FUNCTION_BLOCK FB_WriteRFID
VAR_INPUT
	bAutoNumber				:BOOL;		
	byFirstByteInput		:BYTE;
	bySecondByteInput		:BYTE;
	byLastByteInput			:BYTE;

	bReset					:BOOL;		//reset licznika
END_VAR
VAR_IN_OUT
	bEnable					:BOOL;		//zalczenie bloku
	byIDtoWrite				:BYTE;		//ID do wczytania
END_VAR


VAR_OUTPUT
	byFirstByteOutput		:BYTE;
	bySecondByteOutput		:BYTE;
	byThirdByteOutput		:BYTE;
	byFourthByteOutput		:BYTE;
	byFifthByteOutput		:BYTE;
	byLastByteOutput		:BYTE;
	bDone					:BOOL;		//informacja o prawidlowym zakoczeniu zapisu
	bError					:BOOL;
	iCounterDone			:INT;		//licznik operacji zapisu zakonczonych sukcesem
END_VAR
VAR
	
	iStep: INT;
	tonDelayError	:TON;
END_VAR

IF bReset THEN
	iCounterDone	:=0;
	iStep := 0;
	byFirstByteOutput := byLastByteOutput := 0;
	bReset := FALSE;
END_IF

CASE iStep OF
	0:  //init	
		IF byFirstByteInput = 129 AND bEnable THEN
			bDone:=FALSE; 
			iStep:=10;
		END_IF
	
	10:  //write command
		bySecondByteOutput 	:= 02;
		byThirdByteOutput	:= 00;
		byFourthByteOutput	:= 00;
		byFifthByteOutput 	:= 01;
		byFirstByteOutput := byLastByteOutput := 01;
	
		IF byFirstByteInput = 163 THEN
			iStep := 20;
		ELSIF NOT byFirstByteInput = 163 AND tonDelayError.Q = TRUE THEN
			iStep := 100;
		END_IF
	
	20: //write data
		IF bAutoNumber THEN
			bySecondByteOutput := byIDtoWrite + INT_TO_BYTE(iCounterDone); 
		ELSE
			bySecondByteOutput := byIDtoWrite;
		END_IF
			
		byFirstByteOutput := byLastByteOutput := 65;
		IF byFirstByteInput = 167 THEN
			iStep := 30;
		ELSIF NOT byFirstByteInput = 167 AND tonDelayError.Q = TRUE THEN
			iStep := 100;
		END_IF
	
	30: //check status
		byFirstByteOutput := byLastByteOutput := 0;
		iCounterDone	:= iCounterDone + 1; 
		bDone			:= TRUE; 	
		IF byFirstByteInput = 128 THEN
			iStep := 0;
			byIDtoWrite		:= byIDtoWrite+1;	
		ELSIF NOT byFirstByteInput = 128 AND tonDelayError.Q = TRUE THEN
			iStep := 100;
		END_IF
		bEnable:=FALSE;
	100: // errors
		bError		:= TRUE;
		



END_CASE

END_FUNCTION_BLOCK

(* stored: Version 1.1.0.1, ProductVersion 3.1.4026.13, FileIdentifier 63a4b6d05e9b3b9c12b060e23bc56485882f3c33, FileSignature 7daf9c6d37c078c76c21672664bd1ecadcb83f001698ec7e271a19ce9f484e200f64d6f2fc96a1af96b2467f64b0c499b1ab82cc86b445a642904691cdda37594fbb01e8454857be9d9a1ef66906c1137c0c21bf2b09211ce1d4188f9f5dbae829ad3a788fbfe3c3fdf4f50128dc70bf663c95193885742ba852e101aef0e936de880b6aa6b1930814078a8c0c4093f3d71b79dbc8c7bbc4593d796a8dcbe8c596c24a83adce08586baf7a026b15e626dd6cb8e20b111a60f94aeb14c6e81735276d5b3413379bf3ce389977fd1bd38015545a50ccf18b4d776e5b62bdb0c2e7310947998a4392f935ddaf20f3300321cd21f12790b6ab04d733f2a58e9a08f1
   POU FB_WriteRFID: Id {9e6cc8f6-d4b7-433f-a011-fc44bf01bb2d}, SpecialFunc None *)
